INTERFACE RecipeValue EXTENDS Disposable

{attribute 'monitoring' := 'call'}
PROPERTY Assignment : STRING
GET
END_GET
SET
END_SET
END_PROPERTY

METHOD BuildAndGetAssignmentString : POINTER TO STRING
END_METHOD

METHOD Dispose
VAR_INPUT
END_VAR
END_METHOD

{attribute 'monitoring' := 'call'}
PROPERTY Name : T_MaxString
GET
END_GET
SET
END_SET
END_PROPERTY

END_INTERFACE

(* stored: Version 1.1.0.1
   Itf RecipeValue: Id {10526825-4eae-0cf1-2d65-fc0b8b7d3392}
   Property Assignment: Id {e3fcb79e-b4bc-0931-0f99-2c5b1ddaca8a}
   Get Get: Id {e6672e5d-d30e-00f5-28b4-a62a16f0689a}
   Set Set: Id {3d0135c9-1cba-00dd-09a6-34f535593b08}
   Method BuildAndGetAssignmentString: Id {9fc7466d-b4d0-0591-1c75-00641ec1f548}
   Method Dispose: Id {d2bd2681-d1d5-0d12-285e-6abadc415be7}
   Property Name: Id {b2fc78d9-a141-0fe0-1d41-65176e85faf4}
   Get Get: Id {53c948ac-6637-03c8-11ef-65cec4d00cc8}
   Set Set: Id {5d416326-5b16-0676-365a-3f1166940f69} *)
